{attribute 'qualified_only'}
{attribute 'strict'}
TYPE E_Message_HouseC :
(
	eNoMessage := 0,
	eTooMuchHouseC := 1,
	eErrorHouseC := 2,
	eNoConnectionToBackend := 3
);
END_TYPE

(* stored: Version 1.1.0.1, ProductVersion 3.1.4024.6
   DUT E_Message_HouseC: Id {081a6311-123b-48b0-b4b3-917d5849b6a9} *)
